FUNCTION_BLOCK MAX_LWORD (* IEC 61131-3 LWORD Maximum *)
  (* Standard: 61131-3 *)
  (* Version 0.0, 2004-12-15, JHC, Rockwell Automation, Converted from SRC format. *)
  (* Compiler header: package fb.rt.plc.select; *)
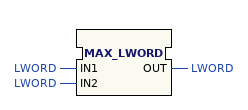
  VAR_INPUT
    IN1 : LWORD;
    IN2 : LWORD;
  END_VAR
  VAR_OUTPUT
    OUT : LWORD; (* MAX(IN1,IN2) *)
  END_VAR
END_FUNCTION_BLOCK
